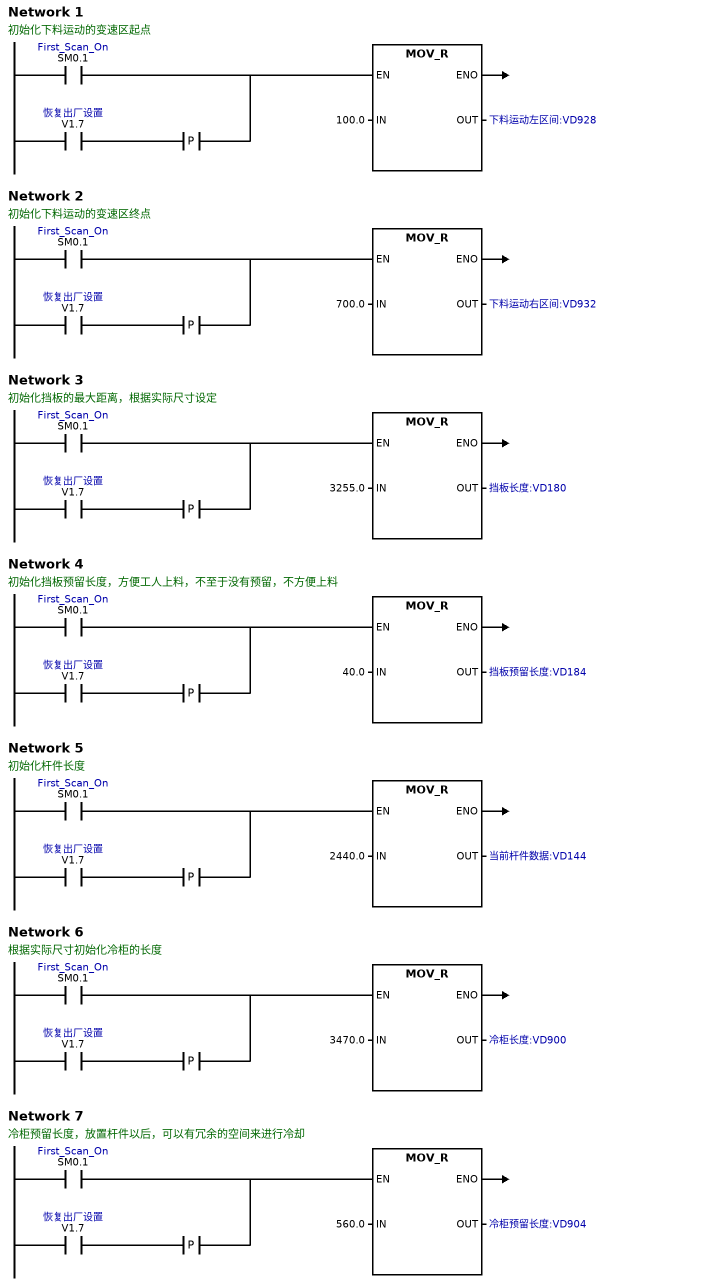
[picture p48: SBR20 networks 1-7]
Network 1
// 初始化下料运动的变速区起点
LD     First_Scan_On:SM0.1
LD     恢复出厂设置:V1.7
EU
OLD
MOVR   100.0, 下料运动左区间:VD928
Network 2
// 初始化下料运动的变速区终点
LD     First_Scan_On:SM0.1
LD     恢复出厂设置:V1.7
EU
OLD
MOVR   700.0, 下料运动右区间:VD932
Network 3
// 初始化挡板的最大距离，根据实际尺寸设定
LD     First_Scan_On:SM0.1
LD     恢复出厂设置:V1.7
EU
OLD
MOVR   3255.0, 挡板长度:VD180
Network 4
// 初始化挡板预留长度，方便工人上料，不至于没有预留，不方便上料
LD     First_Scan_On:SM0.1
LD     恢复出厂设置:V1.7
EU
OLD
MOVR   40.0, 挡板预留长度:VD184
Network 5
// 初始化杆件长度
LD     First_Scan_On:SM0.1
LD     恢复出厂设置:V1.7
EU
OLD
MOVR   2440.0, 当前杆件数据:VD144
Network 6
// 根据实际尺寸初始化冷柜的长度
LD     First_Scan_On:SM0.1
LD     恢复出厂设置:V1.7
EU
OLD
MOVR   3470.0, 冷柜长度:VD900
Network 7
// 冷柜预留长度，放置杆件以后，可以有冗余的空间来进行冷却
LD     First_Scan_On:SM0.1
LD     恢复出厂设置:V1.7
EU
OLD
MOVR   560.0, 冷柜预留长度:VD904
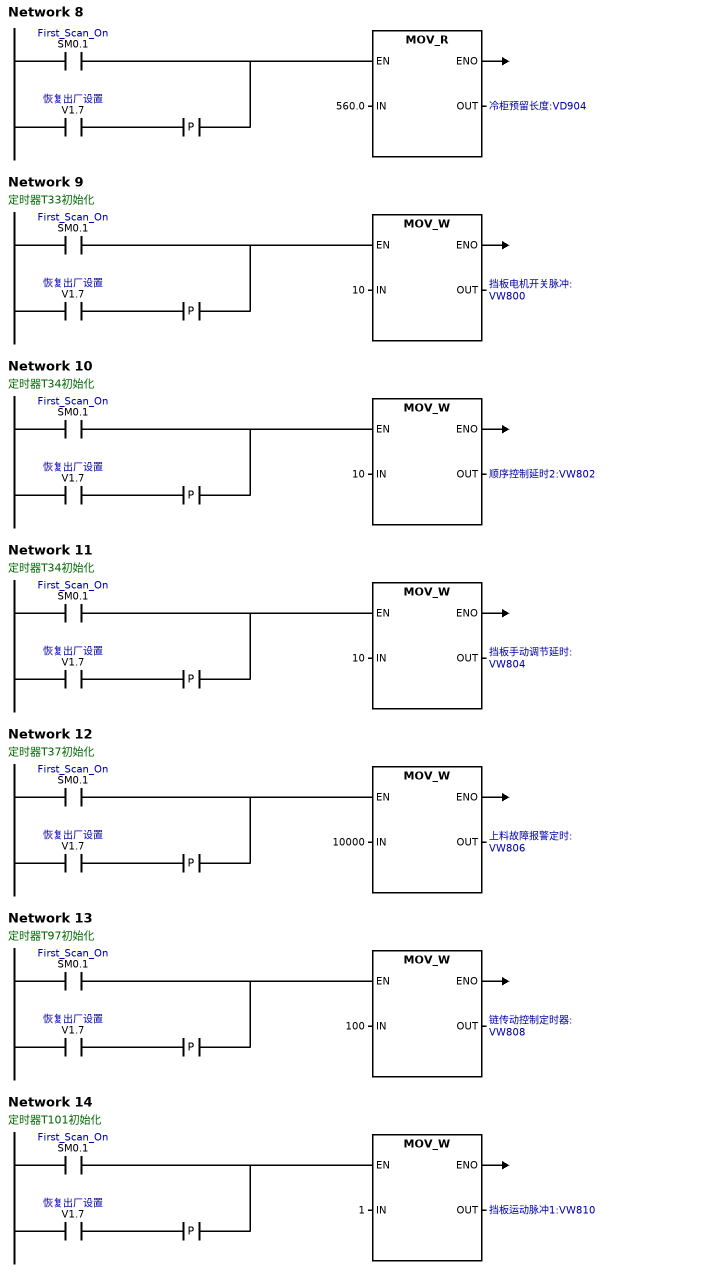
Network 8
LD     First_Scan_On:SM0.1
LD     恢复出厂设置:V1.7
EU
OLD
MOVR   560.0, 冷柜预留长度:VD904
Network 9
// 定时器T33初始化
LD     First_Scan_On:SM0.1
LD     恢复出厂设置:V1.7
EU
OLD
MOVW   10, 挡板电机开关脉冲:VW800
Network 10
// 定时器T34初始化
LD     First_Scan_On:SM0.1
LD     恢复出厂设置:V1.7
EU
OLD
MOVW   10, 顺序控制延时2:VW802
Network 11
// 定时器T34初始化
LD     First_Scan_On:SM0.1
LD     恢复出厂设置:V1.7
EU
OLD
MOVW   10, 挡板手动调节延时:VW804
Network 12
// 定时器T37初始化
LD     First_Scan_On:SM0.1
LD     恢复出厂设置:V1.7
EU
OLD
MOVW   10000, 上料故障报警定时:VW806
Network 13
// 定时器T97初始化
LD     First_Scan_On:SM0.1
LD     恢复出厂设置:V1.7
EU
OLD
MOVW   100, 链传动控制定时器:VW808
Network 14
// 定时器T101初始化
LD     First_Scan_On:SM0.1
LD     恢复出厂设置:V1.7
EU
OLD
MOVW   1, 挡板运动脉冲1:VW810
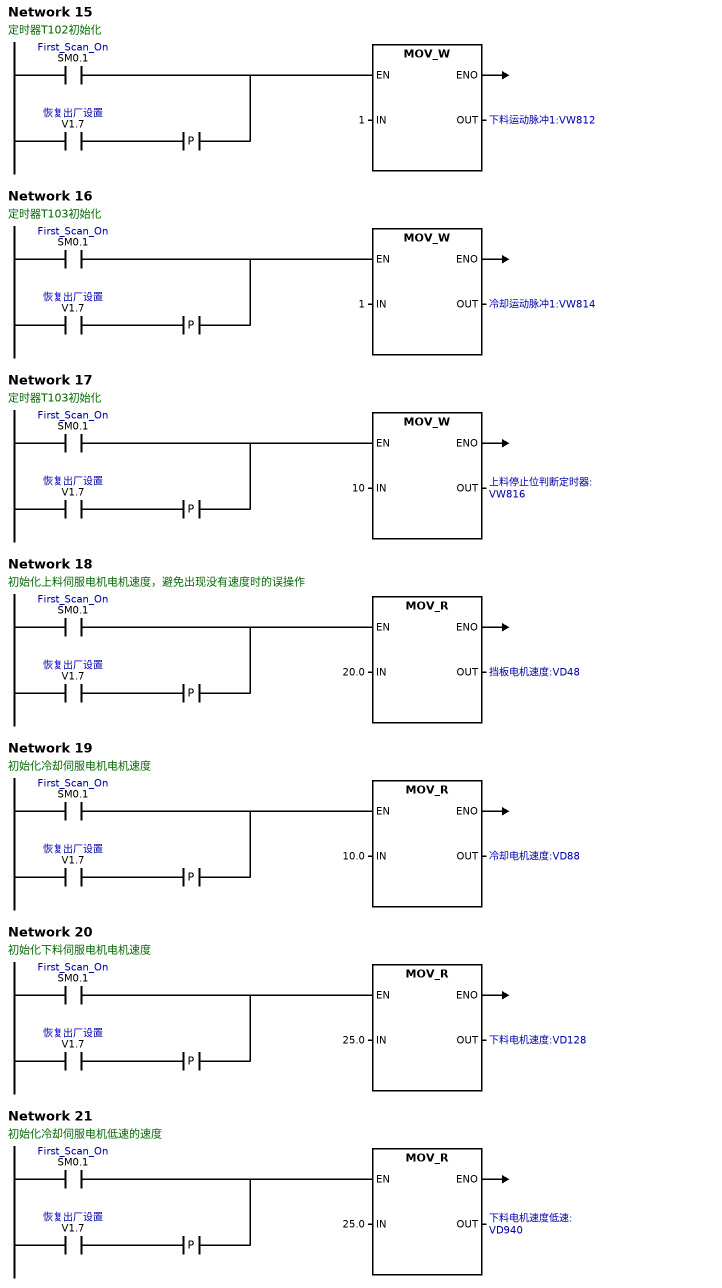
Network 15
// 定时器T102初始化
LD     First_Scan_On:SM0.1
LD     恢复出厂设置:V1.7
EU
OLD
MOVW   1, 下料运动脉冲1:VW812
Network 16
// 定时器T103初始化
LD     First_Scan_On:SM0.1
LD     恢复出厂设置:V1.7
EU
OLD
MOVW   1, 冷却运动脉冲1:VW814
Network 17
// 定时器T103初始化
LD     First_Scan_On:SM0.1
LD     恢复出厂设置:V1.7
EU
OLD
MOVW   10, 上料停止位判断定时器:VW816
Network 18
// 初始化上料伺服电机电机速度，避免出现没有速度时的误操作
LD     First_Scan_On:SM0.1
LD     恢复出厂设置:V1.7
EU
OLD
MOVR   20.0, 挡板电机速度:VD48
Network 19
// 初始化冷却伺服电机电机速度
LD     First_Scan_On:SM0.1
LD     恢复出厂设置:V1.7
EU
OLD
MOVR   10.0, 冷却电机速度:VD88
Network 20
// 初始化下料伺服电机电机速度
LD     First_Scan_On:SM0.1
LD     恢复出厂设置:V1.7
EU
OLD
MOVR   25.0, 下料电机速度:VD128
Network 21
// 初始化冷却伺服电机低速的速度
LD     First_Scan_On:SM0.1
LD     恢复出厂设置:V1.7
EU
OLD
MOVR   25.0, 下料电机速度低速:VD940
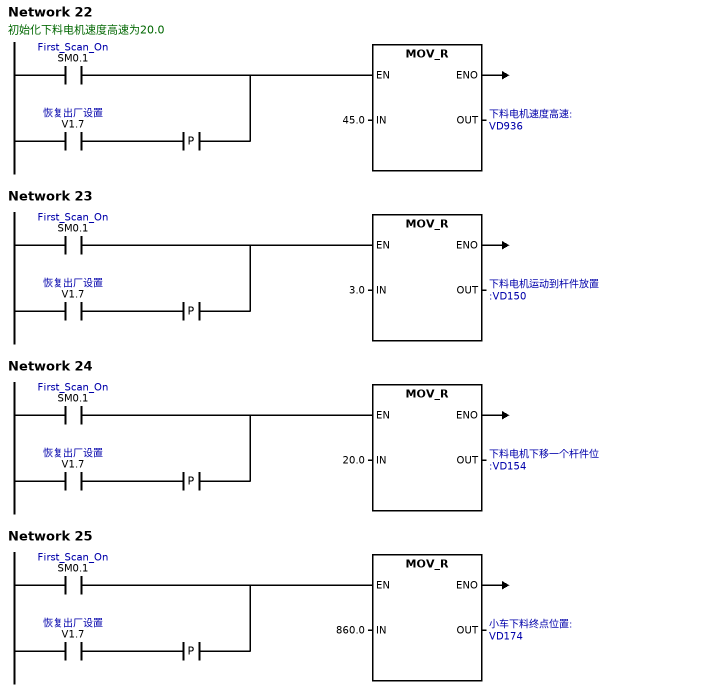
Network 22
// 初始化下料电机速度高速为20.0
LD     First_Scan_On:SM0.1
LD     恢复出厂设置:V1.7
EU
OLD
MOVR   45.0, 下料电机速度高速:VD936
Network 23
LD     First_Scan_On:SM0.1
LD     恢复出厂设置:V1.7
EU
OLD
MOVR   3.0, 下料电机运动到杆件放置:VD150
Network 24
LD     First_Scan_On:SM0.1
LD     恢复出厂设置:V1.7
EU
OLD
MOVR   20.0, 下料电机下移一个杆件位:VD154
Network 25
LD     First_Scan_On:SM0.1
LD     恢复出厂设置:V1.7
EU
OLD
MOVR   860.0, 小车下料终点位置:VD174
END_SUBROUTINE_BLOCK

SUBROUTINE_BLOCK 故障报警:SBR21
TITLE=子程序注释
BEGIN
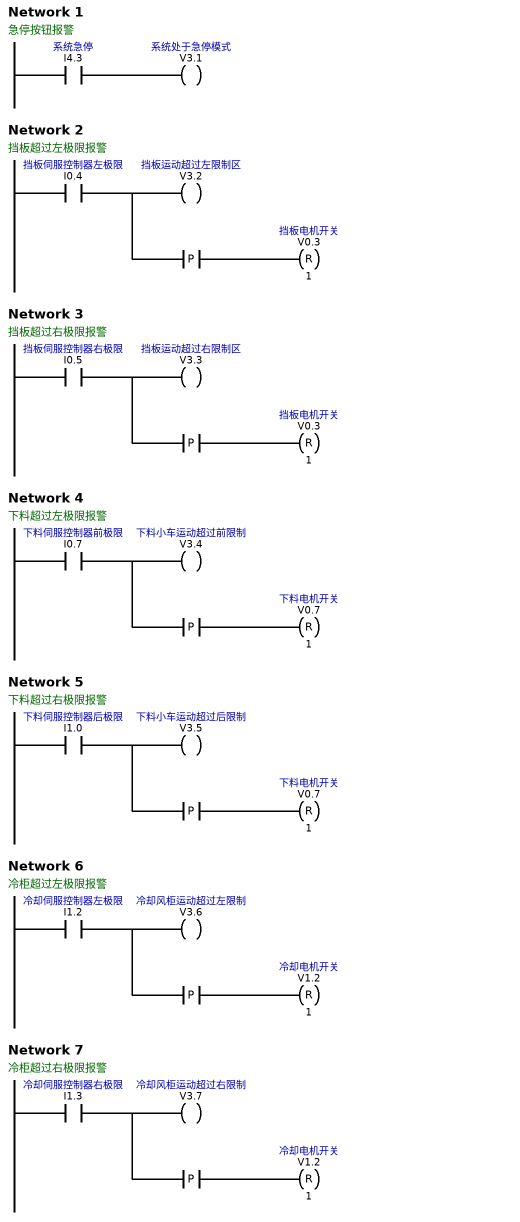
Network 1
// 急停按钮报警
LD     系统急停:I4.3
=      系统处于急停模式:V3.1
Network 2
// 挡板超过左极限报警
LD     挡板伺服控制器左极限:I0.4
=      挡板运动超过左限制区:V3.2
EU
R      挡板电机开关:V0.3, 1
Network 3
// 挡板超过右极限报警
LD     挡板伺服控制器右极限:I0.5
=      挡板运动超过右限制区:V3.3
EU
R      挡板电机开关:V0.3, 1
Network 4
// 下料超过左极限报警
LD     下料伺服控制器前极限:I0.7
=      下料小车运动超过前限制:V3.4
EU
R      下料电机开关:V0.7, 1
Network 5
// 下料超过右极限报警
LD     下料伺服控制器后极限:I1.0
=      下料小车运动超过后限制:V3.5
EU
R      下料电机开关:V0.7, 1
Network 6
// 冷柜超过左极限报警
LD     冷却伺服控制器左极限:I1.2
=      冷却风柜运动超过左限制:V3.6
EU
R      冷却电机开关:V1.2, 1
Network 7
// 冷柜超过右极限报警
LD     冷却伺服控制器右极限:I1.3
=      冷却风柜运动超过右限制:V3.7
EU
R      冷却电机开关:V1.2, 1
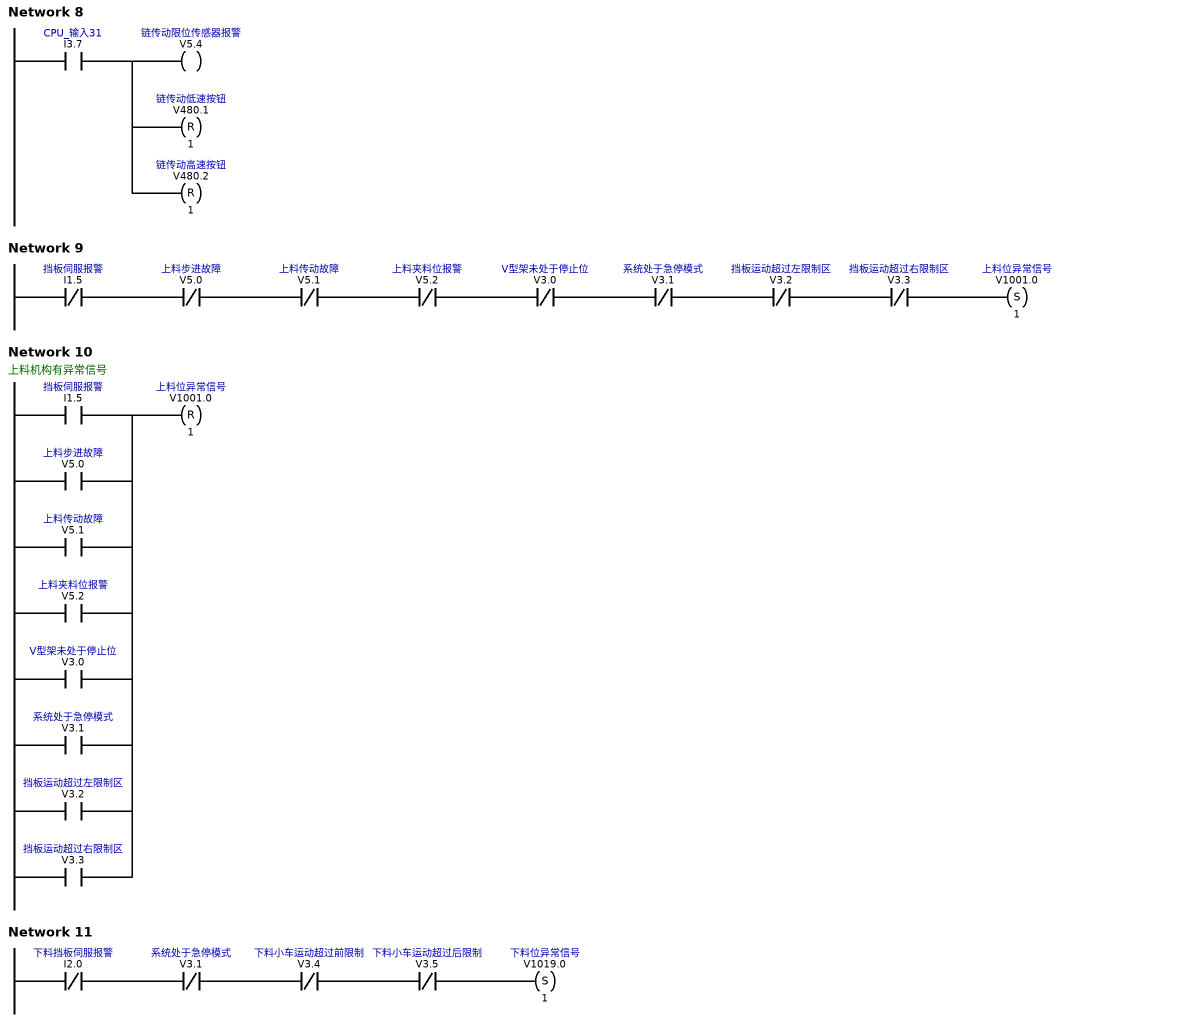
Network 8
LD     CPU_输入31:I3.7
=      链传动限位传感器报警:V5.4
R      链传动低速按钮:V480.1, 1
R      链传动高速按钮:V480.2, 1
Network 9
LDN    挡板伺服报警:I1.5
AN     上料步进故障:V5.0
AN     上料传动故障:V5.1
AN     上料夹料位报警:V5.2
AN     V型架未处于停止位:V3.0
AN     系统处于急停模式:V3.1
AN     挡板运动超过左限制区:V3.2
AN     挡板运动超过右限制区:V3.3
S      上料位异常信号:V1001.0, 1
Network 10
// 上料机构有异常信号
LD     挡板伺服报警:I1.5
O      上料步进故障:V5.0
O      上料传动故障:V5.1
O      上料夹料位报警:V5.2
O      V型架未处于停止位:V3.0
O      系统处于急停模式:V3.1
O      挡板运动超过左限制区:V3.2
O      挡板运动超过右限制区:V3.3
R      上料位异常信号:V1001.0, 1
Network 11
LDN    下料挡板伺服报警:I2.0
AN     系统处于急停模式:V3.1
AN     下料小车运动超过前限制:V3.4
AN     下料小车运动超过后限制:V3.5
S      下料位异常信号:V1019.0, 1
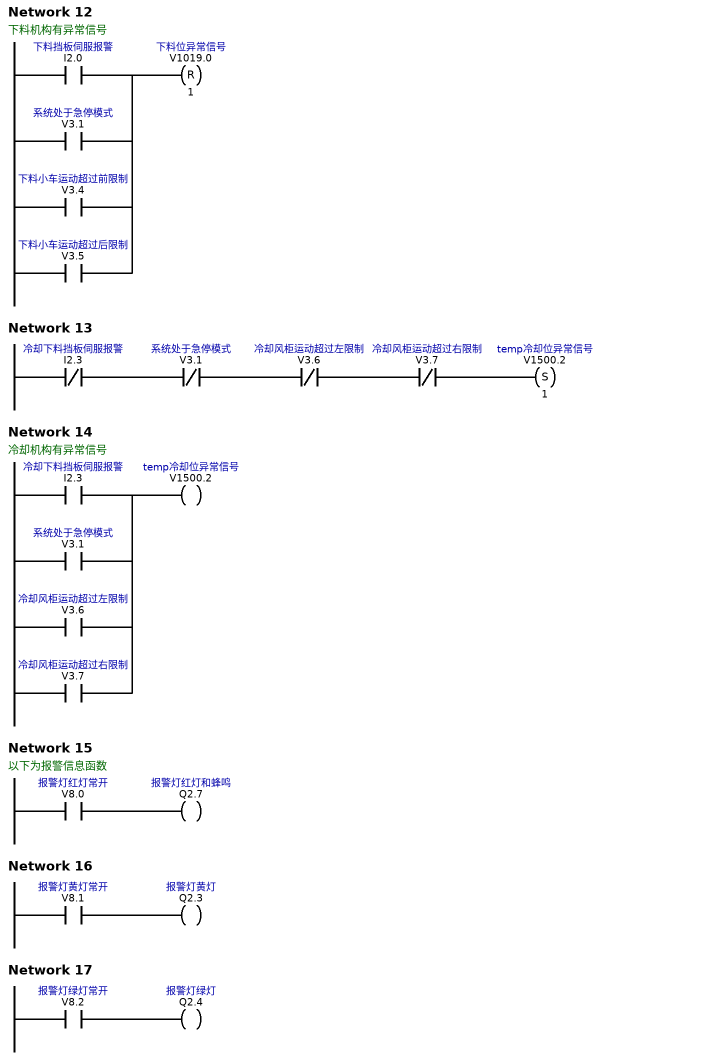
Network 12
// 下料机构有异常信号
LD     下料挡板伺服报警:I2.0
O      系统处于急停模式:V3.1
O      下料小车运动超过前限制:V3.4
O      下料小车运动超过后限制:V3.5
R      下料位异常信号:V1019.0, 1
Network 13
LDN    冷却下料挡板伺服报警:I2.3
AN     系统处于急停模式:V3.1
AN     冷却风柜运动超过左限制:V3.6
AN     冷却风柜运动超过右限制:V3.7
S      temp冷却位异常信号:V1500.2, 1
Network 14
// 冷却机构有异常信号
LD     冷却下料挡板伺服报警:I2.3
O      系统处于急停模式:V3.1
O      冷却风柜运动超过左限制:V3.6
O      冷却风柜运动超过右限制:V3.7
=      temp冷却位异常信号:V1500.2
Network 15
// 以下为报警信息函数
LD     报警灯红灯常开:V8.0
=      报警灯红灯和蜂鸣:Q2.7
Network 16
LD     报警灯黄灯常开:V8.1
=      报警灯黄灯:Q2.3
Network 17
LD     报警灯绿灯常开:V8.2
=      报警灯绿灯:Q2.4
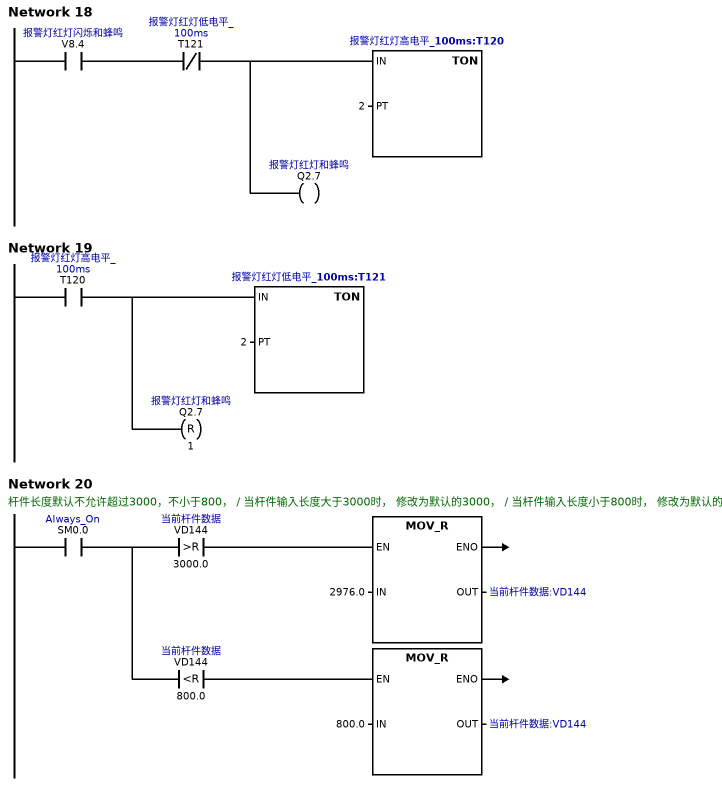
Network 18
LD     报警灯红灯闪烁和蜂鸣:V8.4
AN     报警灯红灯低电平_100ms:T121
TON    报警灯红灯高电平_100ms:T120, 2
=      报警灯红灯和蜂鸣:Q2.7
Network 19
LD     报警灯红灯高电平_100ms:T120
TON    报警灯红灯低电平_100ms:T121, 2
R      报警灯红灯和蜂鸣:Q2.7, 1
Network 20
// 杆件长度默认不允许超过3000，不小于800，
// 当杆件输入长度大于3000时， 修改为默认的3000，
// 当杆件输入长度小于800时， 修改为默认的800
LD     Always_On:SM0.0
LPS
AR>    当前杆件数据:VD144, 3000.0
MOVR   2976.0, 当前杆件数据:VD144
LPP
AR<    当前杆件数据:VD144, 800.0
MOVR   800.0, 当前杆件数据:VD144
END_SUBROUTINE_BLOCK
